TYPE ST_System_FBT_Parameter :
STRUCT
	Temp_Vorl_Max			: REAL;
	Temp_Vorl_Min			: REAL;

	Temp_Warmwasser_Max    : REAL;
	Temp_Warmwasser_Min    : REAL;

	Temp_Kaltwasser_Max    : REAL;
	Temp_Kaltwasser_Min    : REAL;

	Test1: REAL;
	Test2: REAL;
	Test: REAL;


	Kennlinie_Heizung		: ST_Parameter_Kennlinie_Heizung_Kuehlung;
	Kennlinie_Kuehlung		: ST_Parameter_Kennlinie_Heizung_Kuehlung;
	Kennlinie_Tctr			: DINT := 5000;

	Nachtabsenkung_Mo		: ST_Parameter_Nachtabsenkung;
	Nachtabsenkung_Di		: ST_Parameter_Nachtabsenkung;
	Nachtabsenkung_Mi		: ST_Parameter_Nachtabsenkung;
	Nachtabsenkung_Do		: ST_Parameter_Nachtabsenkung;
	Nachtabsenkung_Fr		: ST_Parameter_Nachtabsenkung;
	Nachtabsenkung_Sa		: ST_Parameter_Nachtabsenkung;
	Nachtabsenkung_So		: ST_Parameter_Nachtabsenkung;

	AutoQuittierung			: BOOL := 0;
END_STRUCT
END_TYPE

(* stored: Version 1.1.0.1, ProductVersion 3.1.4024.9
   DUT ST_System_FBT_Parameter: Id {013f9a02-333c-423e-b6b3-0b0512e05e64} *)
